FUNCTION_BLOCK PowerSupply
VAR
	ComHandler : I_CommsTransceiver;
	CommandBuffer : CommandBuffer;
	_targetVoltage : LREAL;
END_VAR

METHOD PUBLIC Beep
VAR
	newCommand : POINTER TO CMD_Beep;
END_VAR
IF NOT CommandBuffer.isFull THEN 
	newCommand := __NEW(CMD_Beep(Comms := THIS^.ComHandler));
	CommandBuffer.Insert(newCommand^); 
END_IF
END_METHOD

METHOD PUBLIC Connect
VAR
	newCommand: POINTER TO CMD_RemoteMode;
END_VAR
IF NOT CommandBuffer.isFull THEN 
	newCommand := __NEW(CMD_RemoteMode(Comms := THIS^.ComHandler));
	CommandBuffer.Insert(newCommand^); 
END_IF
END_METHOD

METHOD PUBLIC CyclicCall
CommandBuffer.CurrentCommand.Execute();
		
IF CommandBuffer.CurrentCommand.isComplete THEN 
	CommandBuffer.Next();
	RETURN;
END_IF
END_METHOD

METHOD PUBLIC Disconnect
VAR
	newCommand: POINTER TO CMD_LocalMode;
END_VAR
IF NOT CommandBuffer.isFull THEN 
	newCommand := __NEW(CMD_LocalMode(Comms := THIS^.ComHandler));
	CommandBuffer.Insert(newCommand^); 
END_IF
END_METHOD

METHOD FB_init : BOOL
VAR_INPUT
	bInitRetains : BOOL; // if TRUE, the retain variables are initialized (warm start / cold start)
	bInCopyCode : BOOL;  // if TRUE, the instance afterwards gets moved into the copy code (online change)
	Comms : I_CommsTransceiver;
END_VAR
THIS^.ComHandler := Comms;
END_METHOD

METHOD PUBLIC QueryTargetVoltage
VAR
	newCommand: POINTER TO CMD_QueryTargetVoltage;
END_VAR
IF NOT CommandBuffer.isFull THEN 
	newCommand := __NEW(CMD_QueryTargetVoltage(Comms := THIS^.ComHandler, ReferenceToResult:=_targetVoltage));
	CommandBuffer.Insert(newCommand^); 
END_IF
END_METHOD

PROPERTY PUBLIC TargetVoltage : LREAL
GET
TargetVoltage := this^._targetVoltage;
END_GET
END_PROPERTY

END_FUNCTION_BLOCK

(* stored: Version 1.1.0.1, ProductVersion 3.1.4024.9
   POU PowerSupply: Id {cf1e44a0-13c6-46f0-b17e-d988703c2722}, SpecialFunc None
   Folder Constructor: Id {f6d2edf1-5226-4dc1-9698-57c0bbb4ba86}
   Folder Properties: Id {da643916-7943-47e4-9942-5954675e5d0f}
   Folder Public: Id {67385631-0e8f-4e72-8a98-cf6f27cc0970}
   Method Beep: Id {586c8e92-565d-45db-af5c-995c8f708a01}
   Method Connect: Id {b601c4c6-4d88-40f0-9695-8ba8bde6a7c6}
   Method CyclicCall: Id {5e4355a5-bcde-4609-931a-21a8ea87d393}
   Method Disconnect: Id {738fa106-00c9-421d-bc11-a6527958d7bc}
   Method FB_init: Id {7503458c-d3f0-4985-9b37-caad344ae25e}
   Method QueryTargetVoltage: Id {9f2e3d82-0eed-4cc8-9ea7-c5bcd432632b}
   Property TargetVoltage: Id {88cee3d8-48b3-4a78-b282-9818ddc679ea}
   Get Get: Id {0ef1798f-2cc7-4d7d-815e-8ab4bc9060c3} *)
